{attribute addProperty BoxType "EP2001-1000-0016"}
{attribute addProperty Id "Group_0AT %Q*Group_5423B5073240Group_1AT %Q*Group_9433FC8D3240WcStateAT %I*WcState_64F6A8C6810InfoDataAT %I*InfoData_192954DE1620"}
{attribute addProperty CRC "842957811"}
{attribute addProperty SizeInBites "88"}
{attribute addProperty SizeInBytes "11"}
TYPE EP2001_62CCD780 :
STRUCT
	{attribute addProperty Name "Group_0"}
	Group_0 : Group_5423B507;
	{attribute addProperty Name "Group_1"}
	Group_1 : Group_9433FC8D;
	{attribute addProperty Name "WcState"}
	WcState : WcState_64F6A8C6;
	{attribute addProperty Name "InfoData"}
	InfoData : InfoData_192954DE;
END_STRUCT
END_TYPE

(* stored: Version 1.2.0.0, ProductVersion 3.1.4024.9
   DUT EP2001_62CCD780: Id {6c7bbc1a-eee0-4793-9d44-12d8da40cead} *)
